// TIA Portal V19 export
FUNCTION_BLOCK "RW_SINAMICS_Par"   // FB160, LAD
TITLE = Read Write Parameter of SINAMICS with TOKEN
// stored: Access Published, MemoryReserve 100, SetENOAutomatically false
   VAR_INPUT
      Enable : Bool;
      ReadWrite : Bool;   // 0=Read, 1=Write
      ParNo : UInt;
      Index : UInt;
      AxisNo : USInt;
      HW_ID : HW_IO;
      TokenChain : Int;
      ValueWriteReal : Real;
      ValueWriteDint : DInt;
   END_VAR
   VAR_OUTPUT
      Done : Bool;
      Error : Bool;
      ValueReadReal : Real;
      ValueReadDint : DInt;
   END_VAR
   VAR
      SinaParaS : SinaParaS;
   END_VAR
   VAR_TEMP
      ReadWriteReq : Bool;
   END_VAR
BEGIN

REGION Network 1 (SCL): Main
   #ReadWriteReq := (#Enable OR #SinaParaS.Busy)
                AND NOT ((#SinaParaS.Done OR #SinaParaS.Error) AND #SinaParaS.Start);

   #SinaParaS.Start := "GetToken"(Enable := #ReadWriteReq , Chain := #TokenChain);

   #SinaParaS(ReadWrite := #ReadWrite,
               Parameter := #ParNo,
               Index := #Index,
               AxisNo := #AxisNo,
               hardwareId := #HW_ID,
               ValueWrite1 := #ValueWriteReal,
               ValueWrite2 := #ValueWriteDint,
               ValueRead1 => #ValueReadReal,
               ValueRead2 => #ValueReadDint);

    #Done := #SinaParaS.Done AND #SinaParaS.Start;
    #Error := #SinaParaS.Error AND #SinaParaS.Start;
END_REGION
END_FUNCTION_BLOCK
